FUNCTION_BLOCK FB_RGBController
VAR
	eLEDColor : eColor;
	iRedLED : INT;
	iGreenLED : INT;
	iBlueLED : INT;
	iWhiteLED : INT;
END_VAR
VAR CONSTANT
	iMAX : INT := 32767;		//Maximum Intensity
	iMIN : INT := 0;			//Off
END_VAR

CASE eLEDColor OF
	eColor.RED:
			iRedLED := iMAX;
			iGreenLED := iMIN;
			iBlueLED := iMIN;
			iWhiteLED := iMIN;
	eColor.GREEN:
			iRedLED := iMIN;
			iGreenLED := iMAX;
			iBlueLED := iMIN;
			iWhiteLED := iMIN;	
	eColor.BLUE:
			iRedLED := iMIN;
			iGreenLED := iMIN;
			iBlueLED := iMAX;	
			iWhiteLED := iMIN;
	eColor.WHITE:
			iRedLED := iMIN;
			iGreenLED := iMIN;
			iBlueLED := iMIN;
			iWhiteLED := iMAX;
END_CASE

RGBController.iRed := iRedLED;
RGBController.iGreen := iGreenLED;
RGBController.iBlue := iBlueLED;
RGBController.iWhite := iWhiteLED;

PROPERTY setLEDColor : eColor
SET
eLEDColor := setLEDColor;
END_SET
END_PROPERTY

END_FUNCTION_BLOCK

(* stored: Version 1.1.0.1, ProductVersion 3.1.4024.12
   POU FB_RGBController: Id {ca565f89-09bf-4fd8-94fd-f485682ef50c}, SpecialFunc None
   Property setLEDColor: Id {e01a2934-0ec9-4d27-bfed-ba0348471b8d}
   Set Set: Id {be286157-1cf5-46db-b1dc-fe4aefc1685d} *)
